// TwinCAT 3 PLC project Untitled1
// ProgramVersion: 3.1.4024.0
// libraries:
//   Tc2_Standard, * (Beckhoff Automation GmbH)
//   Tc2_System, * (Beckhoff Automation GmbH)
//   Tc3_Module, * (Beckhoff Automation GmbH)
// project tree:
//   GVLs/ GVL.TcGVL
//   POUs/ FB_DoorControl.TcPOU, Task_1.TcPOU, Task_2.TcPOU
//   / Task_1_1.TcTTO, Task_2_1.TcTTO
// real-time tasks:
//   TASK Task 1: cycle T#5ms, priority 1, ADS port 350
//   TASK Task 2: cycle T#10ms, priority 2, ADS port 351

CONFIGURATION Untitled1
    RESOURCE PLC ON TwinCAT3
        TASK Task_1_1(INTERVAL := T#5ms, PRIORITY := 1);
        TASK Task_2_1(INTERVAL := T#10ms, PRIORITY := 2);
        PROGRAM Task_1 WITH Task_1_1 : Task_1;
        PROGRAM Task_2 WITH Task_2_1 : Task_2;
    END_RESOURCE
END_CONFIGURATION

// ---- GVLs/GVL.TcGVL
{attribute 'qualified_only'}
VAR_GLOBAL
	bCardPresented : BOOL := FALSE;      // Indicates if a card has been presented
    bElevatorRequest : BOOL := FALSE;    // Indicates if the elevator button is pressed
    bElevatorArrived : BOOL := FALSE;    // Indicates if the elevator has arrived at floor 0
    tDoorCloseDelay : TIME := T#5S;      // Delay time to close the door
    tElevatorMoveTime : TIME := T#10S;   // Time it takes for the elevator to reach floor 0
	bDoorClosed: BOOL;
	bAccessGranted : BOOL := FALSE;
END_VAR

// ---- POUs/Task_1.TcPOU
PROGRAM Task_1
VAR
	fbDoorControl : FB_DoorControl;   // Instance of the door control function block
	bCardPresented: BOOL;
	bAccessGranted: BOOL;
END_VAR

// Card validation and access granting logic
IF bCardPresented THEN
    bAccessGranted := TRUE;           // Grant access if card is presented
    fbDoorControl(bStartTimer := TRUE);
ELSE
    bAccessGranted := FALSE;
    fbDoorControl(bStartTimer := FALSE);
END_IF

// Write the door status to the GVL
GVL.bDoorClosed := fbDoorControl.bDoorClosed;

END_PROGRAM

// ---- POUs/FB_DoorControl.TcPOU
FUNCTION_BLOCK FB_DoorControl
VAR_INPUT
    bStartTimer : BOOL;               // Input to start the timer
END_VAR
VAR_OUTPUT
    bDoorClosed : BOOL;               // Output indicating if the door is closed
END_VAR
VAR
    tmrDoor : TON;                    // Timer to control the door closing delay
	tDoorCloseDelay: TIME;
END_VAR

// Timer logic for door closing
IF bStartTimer THEN
    tmrDoor(IN := TRUE, PT := tDoorCloseDelay);
ELSE
    tmrDoor(IN := FALSE);
END_IF

bDoorClosed := NOT tmrDoor.Q;         // Door is closed when timer is done

END_FUNCTION_BLOCK

// ---- POUs/Task_2.TcPOU
PROGRAM Task_2
VAR
	tmrElevatorMove : TON;                  // Timer for the elevator movement
    bLocalAccessGranted : BOOL := FALSE;    // Local copy of the access granted status
    bLocalElevatorRequest : BOOL := FALSE;  // Local copy of the elevator request status
END_VAR

// Read the GVL variables locally to ensure correct types
bLocalAccessGranted := GVL.bAccessGranted;
bLocalElevatorRequest := GVL.bElevatorRequest;

// Elevator control logic
IF bLocalAccessGranted AND bLocalElevatorRequest THEN
    tmrElevatorMove(IN := TRUE, PT := GVL.tElevatorMoveTime);   // Start the elevator movement timer
ELSE
    tmrElevatorMove(IN := FALSE);
END_IF

// Update elevator status in the GVL
IF tmrElevatorMove.Q THEN
    GVL.bElevatorArrived := TRUE;     // Set TRUE when elevator arrives at floor 0
ELSE
    GVL.bElevatorArrived := FALSE;
END_IF

END_PROGRAM
